(* CoDeSys 2.3 export: OUT_DIG.EXP *)

(* POU 30_Outputs/out_DIG, ST *)
PROGRAM out_DIG
VAR

END_VAR
VAR CONSTANT

END_VAR
(* *)
;
END_PROGRAM
